INTERFACE ICommSeq

PROPERTY EState : E_SocketConnectionState
GET
END_GET
END_PROPERTY

PROPERTY MsgFmtStr : T_MaxString
GET
END_GET
END_PROPERTY

METHOD Run
VAR_INPUT
    msgSend : REFERENCE TO uTelegrammOmronTcp;
    msgRcv  : REFERENCE TO uTelegrammOmronTcp;
END_VAR
END_METHOD

END_INTERFACE

(* stored: Version 1.1.0.1, ProductVersion 3.1.4024.12
   Itf ICommSeq: Id {0288787b-92b2-0ae4-1805-041e52f340d8}
   Property EState: Id {267e7815-fb68-0cbf-2d27-6d4044e081a5}
   Get Get: Id {8a62a295-6512-002a-05f7-8814a800c94f}
   Property MsgFmtStr: Id {1d403324-c97a-07cd-3b35-8cb054c8391e}
   Get Get: Id {8fbd84d7-a95a-0fff-2be2-0fc12f2a33b2}
   Method Run: Id {101d01ee-403e-0903-08ca-3ff7e823f98f} *)
